TYPE CONTROL_PARAMETERS :
STRUCT
	Kp		:	REAL;	
	Ti		:	REAL;
	Td		:	REAL;
	LimLow	:	REAL;
	LimHigh	:	REAL;
	bReverseActing	:	BOOL;
	RST	:	BOOL;	//Reset
END_STRUCT
END_TYPE

(* stored: Version 1.1.0.1, ProductVersion 3.1.4024.3
   DUT CONTROL_PARAMETERS: Id {72424fd5-d91e-4b02-ad3c-a13f31754161} *)
